// TIA Portal V17 export
// export: Created 2025-03-10T13:11:52.0840659Z, ExportSetting WithDefaults, DisplayName Totally Integrated Automation Portal, DisplayVersion V17 Update 8, DisplayName TIA Portal Openness, DisplayVersion V17 Update 8, DisplayName TIA Portal Version Control Interface, DisplayVersion V17, DisplayName SINAMICS Startdrive Advanced, DisplayVersion V17 SP2, DisplayName SINAMICS Startdrive G110M, G120, G120C, G120D, G120P, G115D, DisplayVersion V17 SP2, DisplayName SINAMICS Startdrive G130, G150, S120, S150, SINAMICS MV, S210, DisplayVersion V17 SP2, DisplayName STEP 7 Professional, DisplayVersion V17 Update 8, DisplayName SINUMERIK ONE STEP 7 Toolbox, DisplayVersion V17 Update 12, DisplayName SINUMERIK 840D sl STEP 7 Toolbox, DisplayVersion V17 Update 12, DisplayName STEP 7 Safety, DisplayVersion V17 Update 6, DisplayName WinCC Advanced, DisplayVersion V17 Update 8
VAR_GLOBAL   // PLC tag table "TAGS_SAFETY_IO_PROGRAM"
   SAFE_INPUT_MACH_E_STOP AT %I300.0 : Bool;   // SAFETY INPUT MACHINE EMERGENCY STOP
   SAFE_INPUT_MACHINE_CLOSED AT %M10010.0 : Bool;   // SAFETY INPUT MACHINING SAFETY DOOR
   SAFE_INPUT_UNIT_01_STATION_02_CLOSED AT %I350.0 : Bool;   // SAFETY INPUT UNIT 01 STATION 04 SAFETY DOOR
   SAFE_INPUT_UNIT_01_MAIN_CLOSED AT %I350.1 : Bool;   // SAFETY INPUT UNIT 01 MAIN SAFETY DOOR
   SAFE_INPUT_UNIT_01_STATION_04_CLOSED AT %I350.2 : Bool;   // SAFETY INPUT UNIT 01 STATION 04 SAFETY DOOR
   SAFE_INPUT_UNIT_01_MAINT_CLOSED AT %I350.3 : Bool;   // SAFETY INPUT UNIT 01 MAINTENANCE SAFETY DOOR
   SAFE_INPUT_UNIT_02_STATION_02_CLOSED AT %I360.0 : Bool;   // SAFETY INPUT UNIT 02 STATION 02 SAFETY DOOR
   SAFE_INPUT_UNIT_02_MAIN_CLOSED AT %I360.1 : Bool;   // SAFETY INPUT UNIT 02 MAIN SAFETY DOOR
   SAFE_INPUT_UNIT_02_STATION_04_CLOSED AT %I360.2 : Bool;   // SAFETY INPUT UNIT 02 STATION 04 SAFETY DOOR
   FEEDBACK_OFF_E_STOP_IN AT %I35.5 : Bool;   // FEEDBACK OFF E-STOP INPUT
   FEEDBACK_OFF_E_STOP_RST_STR_IN AT %I35.6 : Bool;   // FEEDBACK OFF E-STOP RESET START INPUT
   FEEDBACK_OFF_SAFETY_DOORS_GANTRY_IN AT %M10030.6 : Bool;   // FEEDBACK OFF SAFETY DOORS FOR GANTRY
   FEEDBACK_OFF_SAFE_DOORS_RST_STR_GANTRY_IN AT %M10030.7 : Bool;   // FEEDBACK OFF SAFETY DOORS FOR GANTRY RESET START INPUT
   FEEDBACK_OFF_POWER_ENABLE_IN AT %I36.4 : Bool;   // FEEDBACK OFF POWER ENABLE
   FEEDBACK_OFF_POWER_ENABLE_RST_STR_IN AT %I36.5 : Bool;   // FEEDBACK OFF POWER ENABLE RESET START INPUT
   HT10_CONNECTED_TO_MAIN_PANEL_MPP483 AT %I41.4 : Bool;   // HT10 CONNECTED TO MAIN PANEL MPP483
   HT10_CONNECTED_TO_PN_PLUS AT %M10040.1 : Bool;   // HT10 CONNECTED TO PN PLUS
   SAFE_OUT_E_STOP_OK AT %Q330.0 : Bool;   // SAFETY OUTPUT EMERGENCY STOP OK
   SAFE_OUT_MCH_GTY_DOOR_LCKD AT %M10050.3 : Bool;   // SAFETY OUTPUT MACHINE TO GANTRY SAFETY DOORS LOCKED
   SAFE_OUT_POWER_ENABLE AT %Q330.3 : Bool;   // SAFETY OUTPUT POWER ENABLED
   SAFE_INPUT_GANTRY_ROBOT_E_STOP AT %M10000.1 : Bool;   // SAFETY INPUT GANTRY ROBOT EMERGENCY STOP
   SAFE_INPUT_ENABLING_DEV AT %I310.3 : Bool;   // SAFETY INPUT ENABLING DEVICE
   SAFE_INPUT_LOAD_UNLOAD_CLOSED AT %M10010.1 : Bool;   // SAFETY INPUT LOAD UNLOAD SAFETY DOOR
   SAFE_INPUT_PHD_CLOSED AT %M10010.2 : Bool;   // SAFETY INPUT PART HANDELING SAFETY DOOR
   SAFE_INPUT_GANTRY_HATCH_CLOSED AT %M10011.7 : Bool;   // SAFETY INPUT GANTRY HATCH DOOR
   SAFE_INPUT_UNIT_01R_CLOSED AT %M10010.7 : Bool;   // SAFETY INPUT UNIT 01R SAFETY DOOR
   SAFE_INPUT_UNIT_01L_CLOSED AT %M10011.0 : Bool;   // SAFETY INPUT UNIT 01L SAFETY DOOR
   SAFE_INPUT_MAINTE_PLATFORM_CLOSED AT %M10011.1 : Bool;   // SAFETY INPUT MAINTENANCE PLATFORM SAFETY DOOR
   SAFE_INPUT_CHIP_CRUSHER_CLOSED AT %M10011.4 : Bool;   // SAFETY INPUT CHIP CRUSER SAFETY DOOR
   SAFE_INPUT_AUTOMATIC_DOOR_01R_CLOSED AT %M10011.5 : Bool;   // SAFETY INPUT AUTOMATIC DOOR CLOSED SIDE 01R
   SAFE_INPUT_ROBOT_CELL_CLOSED AT %M10012.0 : Bool;   // SAFETY INPUT ROBOT CELL SAFETY DOOR
   SAFE_INPUT_AUTO_DOOR_BIMANUAL_1 AT %M10012.1 : Bool;   // SAFETY INPUT AUTOMATIC DOOR BIMANUAL 1
   SAFE_INPUT_AUTO_DOOR_BIMANUAL_2 AT %M10012.2 : Bool;   // SAFETY INPUT AUTOMATIC DOOR BIMANUAL 2
   SAFE_OUT_LASER_SOURCE_ENABLE_WORK_CONDITIONS AT %Q340.0 : Bool;   // SAFE OUT LASER SOURCE ENABLE WORK CONDITIONS
   SAFE_INPUT_SETUP_MODE AT %M10005.1 : Bool;   // SAFETY INPUT SETUP MODE
   FEEDBACK_OFF_LASER_SOURCE_ENABLE_WORK_CONDITIONS_IN AT %I36.6 : Bool;   // FEEDBACK OFF LASER SOURCE ENABLE WORK CONDITIONS IN
   FEEDBACK_OFF_LASER_SOURCE_ENABLE_WORK_CONDITIONS_RST_STR_IN AT %I36.7 : Bool;   // FEEDBACK OFF LASER_SOURCE ENABLE WORK CONDITIONS RST STR IN
   FEEDBACK_OFF_MACHINE_E_STOP_IN AT %M10030.2 : Bool;   // FEEDBACK OFF MACHINE E-STOP INPUT
   FEEDBACK_OFF_MACHINE_E_STOP_RST_STR_IN AT %M10030.3 : Bool;   // FEEDBACK OFF MACHINE E-STOP RESET START INPUT
   SAFE_OUT_MACHINE_E_STOP_OK AT %M10050.1 : Bool;   // SAFETY OUTPUT EMERGENCY STOP OK
   SAFE_INPUT_UNIT_02_MAINT_CLOSED AT %I360.3 : Bool;   // SAFETY INPUT UNIT 02 MAINTENANCE SAFETY DOOR
   SAFE_INPUT_LASER_1_E_STOP AT %I300.1 : Bool;   // SAFE INPUT LASER 1 EMERGENCY STOP
   SAFE_INPUT_LASER_2_E_STOP AT %I300.2 : Bool;   // SAFE INPUT LASER 2 EMERGENCY STOP
   FEEDBACK_OFF_SAFE_DOORS_U01_RST_STR_IN AT %I36.1 : Bool;   // FEEDBACK OFF SAFETY DOORS RESET START INPUT
   FEEDBACK_OFF_SAFETY_DOORS_U01_IN AT %I36.0 : Bool;   // FEEDBACK OFF SAFETY DOORS
   SAFE_OUT_SAFE_DOOR_U01_LCKD AT %Q330.1 : Bool;   // SAFETY OUTPUT SAFETY DOORS LOCKED
   FEEDBACK_OFF_SAFE_DOORS_U02_RST_STR_IN AT %I36.3 : Bool;   // FEEDBACK OFF SAFETY DOORS RESET START INPUT
   SAFE_OUT_SAFE_DOOR_U02_LCKD AT %Q330.2 : Bool;   // SAFETY OUTPUT SAFETY DOORS LOCKED
   FEEDBACK_OFF_SAFETY_DOORS_U02_IN AT %I36.2 : Bool;   // FEEDBACK OFF SAFETY DOORS
   SAFE_INPUT_UNIT_01_OERLIKON_CLOSED AT %M10050.7 : Bool;   // SAFETY INPUT UNIT 01 OERLIKON SAFETY DOOR
   SAFE_INPUT_UNIT_02_OERLIKON_CLOSED AT %M10050.6 : Bool;   // SAFETY INPUT UNIT 02 OERLIKON SAFETY DOOR
   BIMANUAL_2_U01_I AT %I351.1 : Bool;   // BIMANUAL 2 UNIT 01 INPUT
   BIMANUAL_2_U02_I AT %I361.1 : Bool;   // BIMANUAL 2 UNIT 02 INPUT
   BIMANUAL_1_U01_I AT %I351.0 : Bool;   // BIMANUAL 1 UNIT 01 INPUT
   BIMANUAL_1_U02_I AT %I361.0 : Bool;   // BIMANUAL 1 UNIT 02 INPUT
END_VAR
